FUNCTION_BLOCK VALSCAN_250C7D0577BABBFF9 (* Service interface function block type *)
  (* Standard: 61499-2 *)
  (* Version 1.0, 02.07.2012, hoegdan, nxtControl GmbH, Initial Version *)
  PACKAGE Main;
  (* Compiler Cpp nxtControl builtin 1.0 *)
  {SET_ATTRIBUTE(Runtime.FBType.ImplementingType, Runtime.Standard#DYNGEN_VALSCAN)}
  {SET_ATTRIBUTE(Configuration.GenericFBType.InterfaceParams, Runtime.Standard#I:=11;VALUE${I$}:LINT,LINT,LINT,STRING,BOOL,BOOL,BOOL,BOOL,BOOL,BOOL,BOOL)}
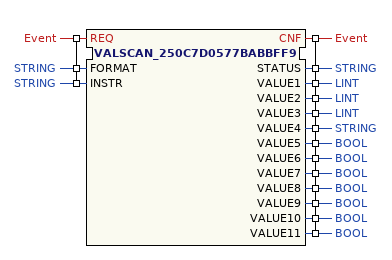
  EVENT_INPUT
    REQ WITH FORMAT, INSTR; (* Request a formatting operation *)
  END_EVENT
  EVENT_OUTPUT
    CNF WITH STATUS, VALUE1, VALUE2, VALUE3, VALUE4, VALUE5, VALUE6, VALUE7, VALUE8, VALUE9, VALUE10, VALUE11; (* Confirms a formattiong operation *)
  END_EVENT
  VAR_INPUT
    FORMAT : STRING; (* Defines a standard C printf like format *)
    INSTR : STRING; (* The input string where the output values are read from *)
  END_VAR
  VAR_OUTPUT
    STATUS : STRING; (* Error information *)
    VALUE1 : LINT; (* A list of values to be read from input string INSTR as defined in parameter FORMAT *)
    VALUE2 : LINT; (* A list of values to be read from input string INSTR as defined in parameter FORMAT *)
    VALUE3 : LINT; (* A list of values to be read from input string INSTR as defined in parameter FORMAT *)
    VALUE4 : STRING; (* A list of values to be read from input string INSTR as defined in parameter FORMAT *)
    VALUE5 : BOOL; (* A list of values to be read from input string INSTR as defined in parameter FORMAT *)
    VALUE6 : BOOL; (* A list of values to be read from input string INSTR as defined in parameter FORMAT *)
    VALUE7 : BOOL; (* A list of values to be read from input string INSTR as defined in parameter FORMAT *)
    VALUE8 : BOOL; (* A list of values to be read from input string INSTR as defined in parameter FORMAT *)
    VALUE9 : BOOL; (* A list of values to be read from input string INSTR as defined in parameter FORMAT *)
    VALUE10 : BOOL; (* A list of values to be read from input string INSTR as defined in parameter FORMAT *)
    VALUE11 : BOOL; (* A list of values to be read from input string INSTR as defined in parameter FORMAT *)
  END_VAR
  EC_STATES
    START;
  END_STATES
END_FUNCTION_BLOCK
